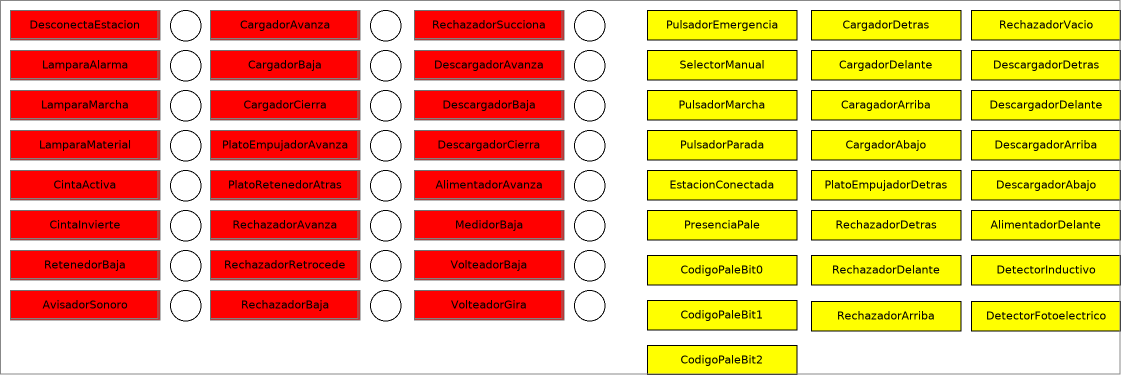
VISUALIZATION Visualization  // 1121x375
    Rectangle (647,170 150x30), "EstacionConectada", colour toggle: MAIN.EstacionConectada
        tap MAIN.EstacionConectada
    Rectangle (647,210 150x30), "PresenciaPale", colour toggle: MAIN.PresenciaPale
        tap MAIN.PresenciaPale
    Rectangle (647,255 150x30), "CodigoPaleBit0", colour toggle: MAIN.CodigoPaleBit0
        tap MAIN.CodigoPaleBit0
    Rectangle (647,300 150x30), "CodigoPaleBit1", colour toggle: MAIN.CodigoPaleBit1
        tap MAIN.CodigoPaleBit1
    Rectangle (647,345 150x30), "CodigoPaleBit2", colour toggle: MAIN.CodigoPaleBit2
        tap MAIN.CodigoPaleBit2
    Button (10,50 150x30), "LamparaAlarma"
        toggle MAIN.LamparaAlarma
    Ellipse (170,50 31x31), colour toggle: MAIN.LamparaAlarma
    Rectangle (647,130 150x30), "PulsadorParada", colour toggle: MAIN.PulsadorParada
        tap MAIN.PulsadorParada
    Rectangle (647,90 150x30), "PulsadorMarcha", colour toggle: MAIN.PulsadorMarcha
        tap MAIN.PulsadorMarcha
    Rectangle (647,50 150x30), "SelectorManual", colour toggle: MAIN.SelectorManual
        toggle MAIN.SelectorManual
    Rectangle (647,10 150x30), "PulsadorEmergencia", colour toggle: MAIN.PulsadorEmergencia
        tap MAIN.PulsadorEmergencia
    Button (10,10 150x30), "DesconectaEstacion"
        toggle MAIN.DesconectaEstacion
    Ellipse (170,10 31x31), colour toggle: MAIN.DesconectaEstacion
    Button (10,130 150x30), "LamparaMaterial"
        toggle MAIN.LamparaMaterial
    Ellipse (170,130 31x31), colour toggle: MAIN.LamparaMaterial
    Button (10,90 150x30), "LamparaMarcha"
        toggle MAIN.LamparaMarcha
    Ellipse (170,90 31x31), colour toggle: MAIN.LamparaMarcha
    Button (10,210 150x30), "CintaInvierte"
        toggle MAIN.CintaInvierte
    Ellipse (170,210 31x31), colour toggle: MAIN.CintaInvierte
    Button (10,170 150x30), "CintaActiva"
        toggle MAIN.CintaActiva
    Ellipse (170,170 31x31), colour toggle: MAIN.CintaActiva
    Button (10,290 150x30), "AvisadorSonoro"
        toggle MAIN.AvisadorSonoro
    Ellipse (170,290 31x31), colour toggle: MAIN.AvisadorSonoro
    Button (10,250 150x30), "RetenedorBaja"
        toggle MAIN.RetenedorBaja
    Ellipse (170,250 31x31), colour toggle: MAIN.RetenedorBaja
    Rectangle (811,170 150x30), "PlatoEmpujadorDetras", colour toggle: MAIN.PlatoEmpujadorDetras
        tap MAIN.PlatoEmpujadorDetras
    Rectangle (811,210 150x30), "RechazadorDetras", colour toggle: MAIN.RechazadorDetras
        tap MAIN.RechazadorDetras
    Rectangle (811,255 150x30), "RechazadorDelante", colour toggle: MAIN.RechazadorDelante
        tap MAIN.RechazadorDelante
    Rectangle (811,130 150x30), "CargadorAbajo", colour toggle: MAIN.CargadorAbajo
        tap MAIN.CargadorAbajo
    Rectangle (811,90 150x30), "CaragadorArriba", colour toggle: MAIN.CargadorArriba
        tap MAIN.CargadorArriba
    Rectangle (811,50 150x30), "CargadorDelante", colour toggle: MAIN.CargadorDelante
        tap MAIN.CargadorDelante
    Rectangle (811,10 150x30), "CargadorDetras", colour toggle: MAIN.CargadorDetras
        tap MIAN.CargadorDetras
    Rectangle (811,301 150x30), "RechazadorArriba", colour toggle: MAIN.RechazadorArriba
        tap MAIN.RechazadorArriba
    Button (210,50 150x30), "CargadorBaja"
        toggle MAIN.CargadorBaja
    Ellipse (370,50 31x31), colour toggle: MAIN.CargadorBaja
    Button (210,10 150x30), "CargadorAvanza"
        toggle MAIN.CargadorAvanza
    Ellipse (370,10 31x31), colour toggle: MAIN.CargadorAvanza
    Button (210,130 150x30), "PlatoEmpujadorAvanza"
        toggle MAIN.PlatoEmpujadorAvanza
    Ellipse (370,130 31x31), colour toggle: MAIN.PlatoEmpujadorAvanza
    Button (210,90 150x30), "CargadorCierra"
        toggle MAIN.CargadorCierra
    Ellipse (370,90 31x31), colour toggle: MAIN.CargadorCierra
    Button (210,210 150x30), "RechazadorAvanza"
        toggle MAIN.RechazadorAvanza
    Ellipse (370,210 31x31), colour toggle: MAIN.RechazadorAvanza
    Button (210,170 150x30), "PlatoRetenedorAtras"
        toggle MAIN.PlatoRetenedorAtras
    Ellipse (370,170 31x31), colour toggle: MAIN.PlatoRetenedorAtras
    Button (210,290 150x30), "RechazadorBaja"
        toggle MAIN.RechazadorBaja
    Ellipse (370,290 31x31), colour toggle: MAIN.RechazadorBaja
    Button (210,250 150x30), "RechazadorRetrocede"
        toggle MAIN.RechazadorRetrocede
    Ellipse (370,250 31x31), colour toggle: MAIN.RechazadorRetrocede
    Rectangle (971,170 150x30), "DescargadorAbajo", colour toggle: MAIN.DescargadorAbajo
        tap MAIN.DescargadorAbajo
    Rectangle (971,210 150x30), "AlimentadorDelante", colour toggle: MAIN.AlimentadorDelante
        tap MAIN.AlimentadorDelante
    Rectangle (971,255 150x30), "DetectorInductivo", colour toggle: MAIN.DetectorInductivo
        tap MAIN.DetectorInductivo
    Rectangle (971,130 150x30), "DescargadorArriba", colour toggle: MAIN.DescargadorArriba
        tap MAIN.DescargadorArriba
    Rectangle (971,90 150x30), "DescargadorDelante", colour toggle: MAIN.DescargadorDelante
        tap MAIN.DescargadorDelante
    Rectangle (971,50 150x30), "DescargadorDetras", colour toggle: MAIN.DescargadorDetras
        tap MAIN.DescargadorDetras
    Rectangle (971,10 150x30), "RechazadorVacio", colour toggle: MAIN.RechazadorVacio
        tap MAIN.RechazadorVacio
    Rectangle (971,301 150x30), "DetectorFotoelectrico", colour toggle: MAIN.DetectorFotoelectrico
        tap MAIN.DetectorFotoelectrico
    Button (414,50 150x30), "DescargadorAvanza"
        toggle MAIN.DescargadorAvanza
    Ellipse (574,50 31x31), colour toggle: MAIN.DescargadorAvanza
    Button (414,10 150x30), "RechazadorSucciona"
        toggle MAIN.RechazadorSucciona
    Ellipse (574,10 31x31), colour toggle: MAIN.RechazadorSucciona
    Button (414,130 150x30), "DescargadorCierra"
        toggle MAIN.DescargadorCierra
    Ellipse (574,130 31x31), colour toggle: MAIN.DescargadorCierra
    Button (414,90 150x30), "DescargadorBaja"
        toggle MAIN.DescargadorBaja
    Ellipse (574,90 31x31), colour toggle: MAIN.DescargadorBaja
    Button (414,210 150x30), "MedidorBaja"
        toggle MAIN.MedidorBaja
    Ellipse (574,210 31x31), colour toggle: MAIN.MedidorBaja
    Button (414,170 150x30), "AlimentadorAvanza"
        toggle MAIN.AlimentadorAvanza
    Ellipse (574,170 31x31), colour toggle: MAIN.AlimentadorAvanza
    Button (414,290 150x30), "VolteadorGira"
        toggle MAIN.VolteadorGira
    Ellipse (574,290 31x31), colour toggle: MAIN.VolteadorGira
    Button (414,250 150x30), "VolteadorBaja"
        toggle MAIN.VolteadorBaja
    Ellipse (574,250 31x31), colour toggle: MAIN.VolteadorBaja
END_VISUALIZATION

(* stored: Version 1.1.0.1, ProductVersion 3.1.4024.12
   Visu Visualization: Id {d673722a-6320-49a9-8529-10ae53f6d6d1} *)
